FUNCTION_BLOCK FB_EntryLogic (* Logique convoyeur entree - SIMPLIFIE v2 *)
  (* Standard: 61499-2 *)
  (* Version 1.1, 20/01/2026, Claude, Schneider Electric, Fix: convoyeur continue meme si bloque *)
  PACKAGE Main;
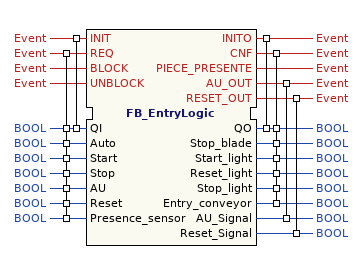
  EVENT_INPUT
    INIT WITH QI; (* Initialization Request *)
    REQ WITH QI, Auto, Start, Stop, AU, Reset, Presence_sensor; (* Normal Execution Request *)
    BLOCK; (* Bloquer entree *)
    UNBLOCK; (* Debloquer entree *)
  END_EVENT
  EVENT_OUTPUT
    INITO WITH QO; (* Initialization Confirm *)
    CNF WITH QO, Stop_blade, Start_light, Reset_light, Stop_light, Entry_conveyor; (* Execution Confirmation *)
    PIECE_PRESENTE; (* Nouvelle piece detectee *)
    AU_OUT WITH AU_Signal; (* Arret urgence active *)
    RESET_OUT WITH Reset_Signal; (* Reset demande *)
  END_EVENT
  VAR_INPUT
    QI : BOOL; (* Input event qualifier *)
    Auto : BOOL;
    Start : BOOL;
    Stop : BOOL;
    AU : BOOL;
    Reset : BOOL;
    Presence_sensor : BOOL;
  END_VAR
  VAR_OUTPUT
    QO : BOOL; (* Output event qualifier *)
    Stop_blade : BOOL;
    Start_light : BOOL;
    Reset_light : BOOL;
    Stop_light : BOOL;
    Entry_conveyor : BOOL;
    AU_Signal : BOOL; (* Signal AU pour autres blocs *)
    Reset_Signal : BOOL; (* Signal Reset pour autres blocs *)
  END_VAR
  VAR
    Presence_prev : BOOL; (* Etat precedent capteur *)
    Blocked : BOOL; (* Entree bloquee *)
  END_VAR
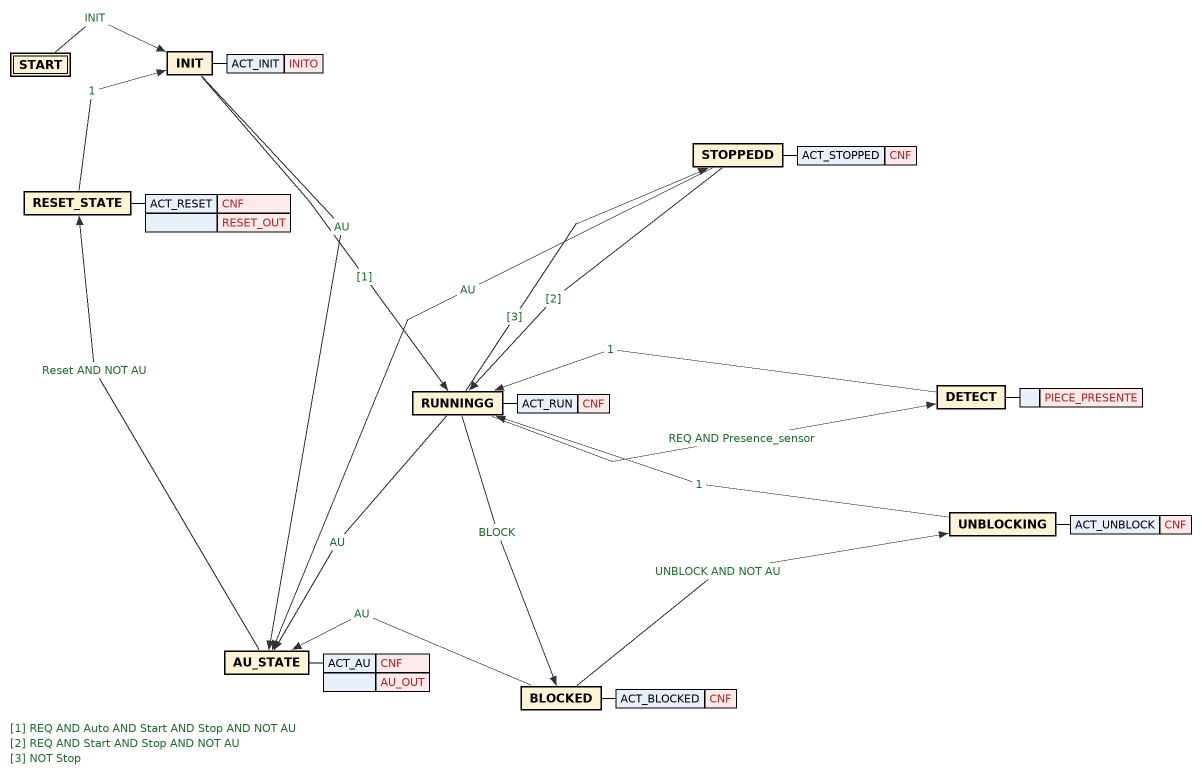
  EC_STATES
    START; (* Initial State *)
    INIT : ACT_INIT -> INITO; (* Initialization *)
    RUNNINGG : ACT_RUN -> CNF; (* Convoyeur en marche *)
    DETECT : -> PIECE_PRESENTE; (* Piece detectee *)
    BLOCKED : ACT_BLOCKED -> CNF; (* Entree bloquee - convoyeur continue *)
    UNBLOCKING : ACT_UNBLOCK -> CNF; (* Deblocage *)
    AU_STATE : ACT_AU -> CNF, -> AU_OUT; (* Arret urgence *)
    RESET_STATE : ACT_RESET -> CNF, -> RESET_OUT; (* Reset *)
    STOPPEDD : ACT_STOPPED -> CNF; (* Arrete *)
  END_STATES
  EC_TRANSITIONS
    START TO INIT := INIT;
    INIT TO RUNNINGG := REQ AND Auto AND Start AND Stop AND NOT AU;
    RUNNINGG TO DETECT := REQ AND Presence_sensor;
    DETECT TO RUNNINGG := 1;
    RUNNINGG TO BLOCKED := BLOCK;
    BLOCKED TO UNBLOCKING := UNBLOCK AND NOT AU;
    UNBLOCKING TO RUNNINGG := 1;
    RUNNINGG TO AU_STATE := AU;
    BLOCKED TO AU_STATE := AU;
    AU_STATE TO RESET_STATE := Reset AND NOT AU;
    RESET_STATE TO INIT := 1;
    RUNNINGG TO STOPPEDD := NOT Stop;
    STOPPEDD TO RUNNINGG := REQ AND Start AND Stop AND NOT AU;
    STOPPEDD TO AU_STATE := AU;
    INIT TO AU_STATE := AU;
  END_TRANSITIONS
  ALGORITHM ACT_INIT IN ST: (* Initialization *)
QO := TRUE;
Entry_conveyor := FALSE;
Stop_blade := FALSE;
Start_light := FALSE;
Reset_light := TRUE;
Stop_light := FALSE;
Presence_prev := FALSE;
Blocked := FALSE;
AU_Signal := FALSE;
Reset_Signal := FALSE;
  END_ALGORITHM
  ALGORITHM ACT_RUN IN ST: (* Convoyeur en marche *)
(* Convoyeur TOUJOURS en marche *)
Entry_conveyor := TRUE;
Stop_blade := FALSE;
Start_light := TRUE;
Reset_light := FALSE;
Stop_light := FALSE;
Presence_prev := Presence_sensor;
  END_ALGORITHM
  ALGORITHM ACT_BLOCKED IN ST: (* Entree bloquee *)
(* Bloquer entree - piece en cours deja sur exit conveyor *)
Blocked := TRUE;
Entry_conveyor := FALSE;  (* Arreter convoyeur entree *)
Stop_blade := TRUE;       (* Lame levee *)
Start_light := TRUE;
Reset_light := FALSE;
Stop_light := FALSE;
Presence_prev := Presence_sensor;
  END_ALGORITHM
  ALGORITHM ACT_UNBLOCK IN ST: (* Debloquer entree *)
(* Debloquer - baisser la lame *)
Blocked := FALSE;
Entry_conveyor := TRUE;
Stop_blade := FALSE;
Start_light := TRUE;
Reset_light := FALSE;
Stop_light := FALSE;
Presence_prev := Presence_sensor;
  END_ALGORITHM
  ALGORITHM ACT_AU IN ST: (* Arret urgence *)
(* Tout arreter immediatement *)
AU_Signal := TRUE;
Reset_Signal := FALSE;
Blocked := FALSE;
Entry_conveyor := FALSE;
Stop_blade := TRUE;
Start_light := FALSE;
Reset_light := TRUE;
Stop_light := TRUE;
Presence_prev := FALSE;
  END_ALGORITHM
  ALGORITHM ACT_RESET IN ST: (* Reset *)
(* Remettre a zero *)
AU_Signal := FALSE;
Reset_Signal := TRUE;
Blocked := FALSE;
Entry_conveyor := FALSE;
Stop_blade := FALSE;
Start_light := FALSE;
Reset_light := TRUE;
Stop_light := FALSE;
Presence_prev := FALSE;
  END_ALGORITHM
  ALGORITHM ACT_STOPPED IN ST: (* Arrete proprement *)
(* Usine arretee *)
Blocked := FALSE;
Entry_conveyor := FALSE;
Stop_blade := FALSE;
Start_light := FALSE;
Reset_light := FALSE;
Stop_light := TRUE;
Presence_prev := FALSE;
  END_ALGORITHM
END_FUNCTION_BLOCK
